PROGRAM MAIN
VAR
	aEvent : ARRAY[1..100] OF ST_Event;
	sTempString : STRING(255);
	
	nReturnGreater : INT;
	nReturnSmaller : INT;
	
	UpdateEventTimestam : ST_Event;
	aBoolean : BOOL := FALSE;
END_VAR

IF NOT aBoolean THEN
	sTempString := aEvent[33].sEventText;
	
	Greater_Smaller(nNumber1 := 8,
		nNumber2 := 15,
		nGreater => nReturnGreater,
		nSmaller => nReturnSmaller);
		
	UpdateEventTimestampWithSystemTime(stEvent := UpdateEventTimestam);
	aBoolean := TRUE;
END_IF

END_PROGRAM

(* stored: Version 1.1.0.1, ProductVersion 3.1.4024.12
   POU MAIN: Id {8333e720-6ccd-401f-8b59-18721b58bade}, SpecialFunc None *)
